(* PLC project Unnamed, Unknown Unnamed 1 *)
(* stored: creationDateTime 2021-09-05T15:38:12, modificationDateTime 2021-10-30T17:49:12 *)

PROGRAM program0
  VAR
    I1 : BOOL;
    I2 : BOOL;
    Q1 : BOOL;
    Q2 : BOOL;
    Q3 : BOOL;
  END_VAR

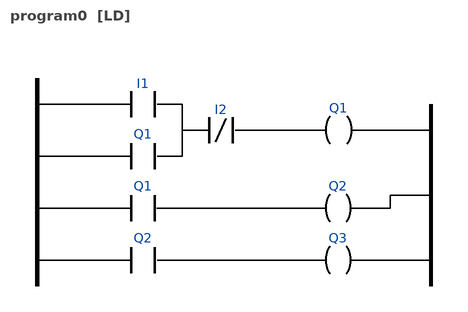
(* LD diagram, written out as Structured Text *)
Q1 := (Q1 OR I1) AND NOT I2;
Q2 := Q1;
Q3 := Q2;
END_PROGRAM

CONFIGURATION Config0
  RESOURCE Res0 ON PLC
    TASK task0(INTERVAL := T#20ms, PRIORITY := 0);
    PROGRAM instance0 WITH task0 : program0;
  END_RESOURCE
END_CONFIGURATION
